// TIA Portal V20 export
TYPE "LWONIK_typeScrapBox"
// stored: Access Published
   STRUCT
      command { S7_SetPoint := 'True'} : "LWONIK_typeScrapBoxCommand";
      monitoring { S7_SetPoint := 'True'} : "LWONIK_typeScrapBoxMonitoring";
   END_STRUCT;
END_TYPE
